// TwinCAT 3 PLC project interlock
// ProgramVersion: 3.1.4023.0
// libraries:
//   VisuElemBase, * (System)
//   Tc2_Standard, * (Beckhoff Automation GmbH)
//   Tc2_System, * (Beckhoff Automation GmbH)
//   Tc3_Module, * (Beckhoff Automation GmbH)
//   Visu Interfaces,newest,System
//   VisuSymbols,3.5.10.0,System
// project tree:
//   / GlobalTextList.TcGTLO, PlcTask.TcTTO, VisualizationManager.TcVMO (not stored), VISU_TASK.TcTTO
//   GVLs/ GVL_ver.TcGVL
//   POUs/ FB_IKR270.TcPOU, FB_KJL300.TcPOU, FB_PBR260.TcPOU, GCC1.TcPOU, GCC2.TcPOU, LadderLogic.TcPOU, LadderLogic_1.TcPOU, MAIN.TcPOU, FB_TCP.TcPOU, VGC1.TcPOU, PTM1.TcPOU, VCC2.TcPOU, VCC3.TcPOU, VGC0.TcPOU
//   VISUs/ Vacuum.TcVIS
// real-time tasks:
//   TASK PlcTask: cycle T#10ms, priority 20, ADS port 350
//   TASK VISU_TASK: cycle T#200000us, priority 30, ADS port 351
// I/O:
//   DEVICE Device 1 (EtherCAT), AmsNetId 5.46.196.210.2.1
//     Term 1 (EK1200) [EK1200-5000 EtherCAT Power supply (2A E-Bus)]
//       Term 2 (EL9210) [EL9210 Power Supplier with LED (24V, Fuse, Diagnostics)]
//       Term 3 (EL3104) [EL3104 4Ch. Ana. Input +/-10V Diff.]
//       Term 4 (EL2004) [EL2004 4Ch. Dig. Output 24V, 0.5A]
//       Term 5 (EL2624) [EL2624 4Ch. Relay Output, NO (125V AC / 30V DC)]
//       Term 6 (EL1104) [EL1104 4Ch. Dig. Input 24V, 3ms, Sensor Power]
//       Term 7 (EL1104) [EL1104 4Ch. Dig. Input 24V, 3ms, Sensor Power]
//       Term 8 (EL2004) [EL2004 4Ch. Dig. Output 24V, 0.5A]
//       Term 9 (EL1104) [EL1104 4Ch. Dig. Input 24V, 3ms, Sensor Power]
//       Term 10 (EL2624) [EL2624 4Ch. Relay Output, NO (125V AC / 30V DC)]
//       Term 11 (EL1104) [EL1104 4Ch. Dig. Input 24V, 3ms, Sensor Power]
//       Term 12 (EL1104) [EL1104 4Ch. Dig. Input 24V, 3ms, Sensor Power]
//       Term 13 (EL2004) [EL2004 4Ch. Dig. Output 24V, 0.5A]
//       Term 14 (EL6022) [EL6022 Interface 2Ch. (RS422/485)]
//       Term 15 (EL6022) [EL6022 Interface 2Ch. (RS422/485)]
//       Term 16 (EK1110) [EK1110 EtherCAT extension]
//   DEVICE Device 3 (CX9020-0115-M310), AmsNetId 5.46.196.210.4.1
//   DEVICE Device 4 (NOV-DP-RAM)
// variable links:
//   interlock Instance <-> Device 1 (EtherCAT)/Term 1 (EK1200)/Term 10 (EL2624)
//     PlcTask Outputs/GVL_ver.VCC2_q_xOPN_DO <-> Channel 1/Output
//   interlock Instance <-> Device 1 (EtherCAT)/Term 1 (EK1200)/Term 12 (EL1104)
//     PlcTask Inputs/GVL_ver.PTM1_i_xAtSpd <-> Channel 1/Input
//     PlcTask Inputs/GVL_ver.PTM1_i_xFaultNC <-> Channel 3/Input
//     PlcTask Inputs/GVL_ver.PTM1_i_xRemote <-> Channel 2/Input
//   interlock Instance <-> Device 1 (EtherCAT)/Term 1 (EK1200)/Term 13 (EL2004)
//     PlcTask Outputs/GVL_ver.PTM1_q_PumpingStation <-> Channel 2/Output
//     PlcTask Outputs/GVL_ver.PTM1_q_RunDO <-> Channel 1/Output
//     PlcTask Outputs/GVL_ver.PTM1_q_xRemote <-> Channel 3/Output
//   interlock Instance <-> Device 1 (EtherCAT)/Term 1 (EK1200)/Term 3 (EL3104)
//     PlcTask Inputs/GVL_ver.GCC1AO <-> AI Standard Channel 1/Value
//     PlcTask Inputs/GVL_ver.GCC2AO <-> AI Standard Channel 2/Value
//   interlock Instance <-> Device 1 (EtherCAT)/Term 1 (EK1200)/Term 4 (EL2004)
//     PlcTask Outputs/GVL_ver.GCC1_xHV_DIS <-> Channel 2/Output
//     PlcTask Outputs/GVL_ver.GCC2_xHV_DIS <-> Channel 4/Output
//   interlock Instance <-> Device 1 (EtherCAT)/Term 1 (EK1200)/Term 6 (EL1104)
//     PlcTask Inputs/GVL_ver.VGC0_i_xClsLS <-> Channel 4/Input
//     PlcTask Inputs/GVL_ver.VGC1_i_xClsLS <-> Channel 3/Input
//     PlcTask Inputs/GVL_ver.VGC0_i_xOpnLS <-> Channel 2/Input
//     PlcTask Inputs/GVL_ver.VGC1_i_xOpnLS <-> Channel 1/Input
//   interlock Instance <-> Device 1 (EtherCAT)/Term 1 (EK1200)/Term 7 (EL1104)
//     PlcTask Inputs/GVL_ver.VCC3_i_xClsLS <-> Channel 4/Input
//     PlcTask Inputs/GVL_ver.VCC3_i_xOpnLS <-> Channel 2/Input
//   interlock Instance <-> Device 1 (EtherCAT)/Term 1 (EK1200)/Term 8 (EL2004)
//     PlcTask Outputs/GVL_ver.VCC3_q_xOPN_DO <-> Channel 4/Output
//     PlcTask Outputs/GVL_ver.VGC0_q_xOPN_DO <-> Channel 3/Output
//     PlcTask Outputs/GVL_ver.VGC1_q_xOPN_DO <-> Channel 1/Output
//   interlock Instance <-> Device 1 (EtherCAT)/Term 1 (EK1200)/Term 9 (EL1104)
//     PlcTask Inputs/GVL_ver.VCC2_i_xClsLS <-> Channel 2/Input
//     PlcTask Inputs/GVL_ver.VCC2_i_xOpnLS <-> Channel 1/Input

CONFIGURATION interlock
    RESOURCE PLC ON TwinCAT3
        TASK PlcTask(INTERVAL := T#10ms, PRIORITY := 20);
        TASK VISU_TASK(INTERVAL := T#200000us, PRIORITY := 30);
        PROGRAM MAIN WITH PlcTask : MAIN;
        PROGRAM VisuElems_Visu_Prg WITH VISU_TASK : VisuElems.Visu_Prg;
    END_RESOURCE
END_CONFIGURATION

// ---- GVLs/GVL_ver.TcGVL
{attribute 'qualified_only'}
VAR_GLOBAL
	V0OPENREQ AT %I*:BOOL;
	V1BYPASS AT %I*:BOOL;
	V2OPENREQ AT %I*:BOOL;
	V3OPENREQ AT %I*:BOOL;
	V4OPENREQ AT %I*:BOOL;
	PTM1STARTREQ AT %I*:BOOL;
	PTM2STARTREQ AT %I*:BOOL;
	PTM3STARTREQ AT %I*:BOOL;
	GCC1ONREQ AT %I*:BOOL;
	GCC2ONREQ AT %I*:BOOL;
	GCC1AO AT %I*:INT;
	GCC2AO AT %I*:INT;

	VGC0OPENREQ AT %I*:BOOL;
	VGC1OPENREQ AT %I*:BOOL;
	VCC2_r_OPENREQ AT %I*:BOOL;
	VCC3_r_OPENREQ AT %I*:BOOL;
	
	PTM1_q_RunDO AT%Q*: BOOL; // Start/Stop for TC110 link this output to the Pumping station bit -3-
    PTM1_q_PumpingStation AT%Q*: BOOL; // Start/Stop interlock -4-
    PTM1_q_xRemote AT%Q*: BOOL; // Remote Priority -14-
    PTM1_i_xAtSpd AT%I*: BOOL; // Normaml operation when true -8-
    PTM1_i_xRemote AT%I*: BOOL; // Remote Priority RBV -23-
	PTM1_i_xFaultNC AT%I*: BOOL; // Error -9-
	
    PTM2_q_RunDO AT%Q*: BOOL; // Start/Stop for TC110 link this output to the Pumping station bit -3-
    PTM2_q_PumpingStation AT%Q*: BOOL; // Start/Stop interlock -4-
    PTM2_q_xRemote AT%Q*: BOOL; // Remote Priority -14-
    PTM2_i_xAtSpd AT%I*: BOOL; // Normaml operation when true -8-
    PTM2_i_xRemote AT%I*: BOOL; // Remote Priority RBV -23-
	PTM2_i_xFaultNC AT%I*: BOOL; // Error -9-
	
	PTM3_q_RunDO AT%Q*: BOOL; // Start/Stop for TC110 link this output to the Pumping station bit -3-
    PTM3_q_PumpingStation AT%Q*: BOOL; // Start/Stop interlock -4-
    PTM3_q_xRemote AT%Q*: BOOL; // Remote Priority -14-
    PTM3_i_xAtSpd AT%I*: BOOL; // Normaml operation when true -8-
    PTM3_i_xRemote AT%I*: BOOL; // Remote Priority RBV -23-
	PTM3_i_xFaultNC AT%I*: BOOL; // Error -9-
	
	VGC0_q_xOPN_DO AT%Q*: BOOL; //24V open/close
	VGC0_i_xOpnLS AT%I*  : BOOL; //Open position SW
    VGC0_i_xClsLS AT%I*  : BOOL; //Close position SW
	VGC0_i_xUpstream_OK  AT%Q*  : BOOL;
	VGC0_i_xDwstream_OK  AT%Q*  : BOOL;
	
	VGC1_q_xOPN_DO AT%Q*: BOOL; //24V open/close
	VGC1_i_xOpnLS AT%I*  : BOOL; //Open position SW
    VGC1_i_xClsLS AT%I*  : BOOL; //Close position SW
	VGC1_i_xUpstream_OK  AT%Q*  : BOOL;
	VGC1_i_xDwstream_OK  AT%Q*  : BOOL;
    
    VCC2_q_xOPN_DO AT%Q*: BOOL; //24V open/close
	VCC2_i_xOpnLS AT%I*  : BOOL; //Open position SW
    VCC2_i_xClsLS AT%I*  : BOOL; //Close position SW
    
    VCC3_q_xOPN_DO AT%Q*: BOOL; //24V open/close
	VCC3_i_xOpnLS AT%I*  : BOOL; //Open position SW
    VCC3_i_xClsLS AT%I*  : BOOL; //Close position SW
    
    GCC1_rPRESS AT%Q* : REAL; //This is the human-readable pressure
    GCC1_xPRESS_OK AT%Q*: BOOL;
	GCC1_xHV_DIS AT %Q* : BOOL;
	
	GCC2_rPRESS AT%Q*: REAL; //This is the human-readable pressure
    GCC2_xPRESS_OK AT%Q*: BOOL;
	GCC2_xHV_DIS AT %Q* : BOOL;

END_VAR

// ---- POUs/MAIN.TcPOU
PROGRAM MAIN
VAR
END_VAR

GVL_ver.GCC2_xHV_DIS:=TRUE;
LadderLogic();
FB_KJL300();
FB_PBR260();
FB_TCP();

END_PROGRAM

// ---- POUs/LadderLogic.TcPOU
PROGRAM LadderLogic
VAR
	ExternalILK: BOOL;
END_VAR

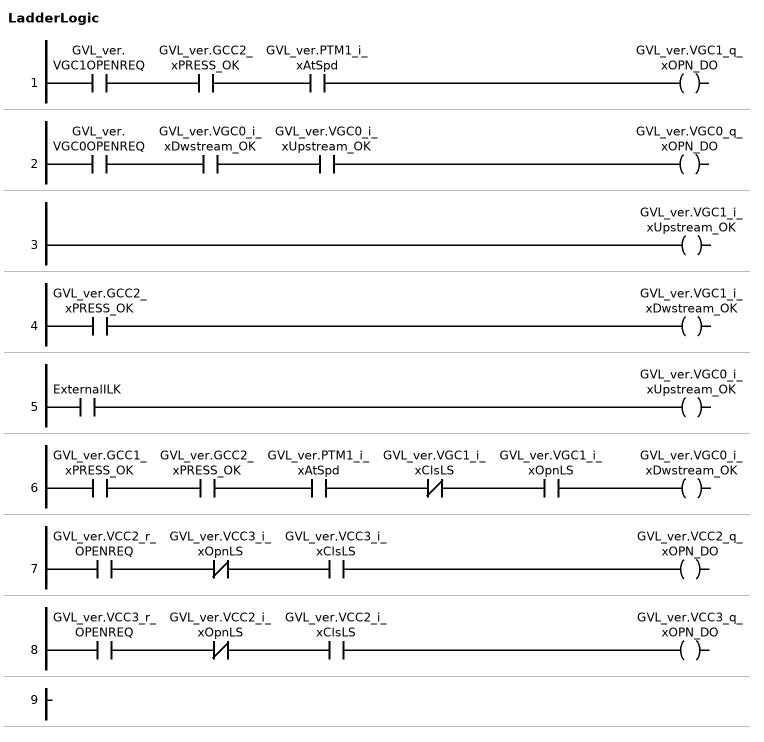
// NETWORK 1
GVL_ver.VGC1_q_xOPN_DO := GVL_ver.VGC1OPENREQ AND GVL_ver.GCC2_xPRESS_OK AND GVL_ver.PTM1_i_xAtSpd;

// NETWORK 2
GVL_ver.VGC0_q_xOPN_DO := GVL_ver.VGC0OPENREQ AND GVL_ver.VGC0_i_xDwstream_OK AND GVL_ver.VGC0_i_xUpstream_OK;

// NETWORK 3
GVL_ver.VGC1_i_xUpstream_OK := TRUE;

// NETWORK 4
GVL_ver.VGC1_i_xDwstream_OK := GVL_ver.GCC2_xPRESS_OK;

// NETWORK 5
GVL_ver.VGC0_i_xUpstream_OK := ExternalILK;

// NETWORK 6
GVL_ver.VGC0_i_xDwstream_OK := GVL_ver.GCC1_xPRESS_OK AND GVL_ver.GCC2_xPRESS_OK AND GVL_ver.PTM1_i_xAtSpd AND NOT GVL_ver.VGC1_i_xClsLS AND GVL_ver.VGC1_i_xOpnLS;

// NETWORK 7
GVL_ver.VCC2_q_xOPN_DO := GVL_ver.VCC2_r_OPENREQ AND NOT GVL_ver.VCC3_i_xOpnLS AND GVL_ver.VCC3_i_xClsLS;

// NETWORK 8
GVL_ver.VCC3_q_xOPN_DO := GVL_ver.VCC3_r_OPENREQ AND NOT GVL_ver.VCC2_i_xOpnLS AND GVL_ver.VCC2_i_xClsLS;

// NETWORK 9

END_PROGRAM

// ---- POUs/FB_KJL300.TcPOU
PROGRAM FB_KJL300
VAR
	AO:INT;
	rPRESS:REAL;
	xPRESS_OK:BOOL;
	xHV_DIS:BOOL:=TRUE;
END_VAR

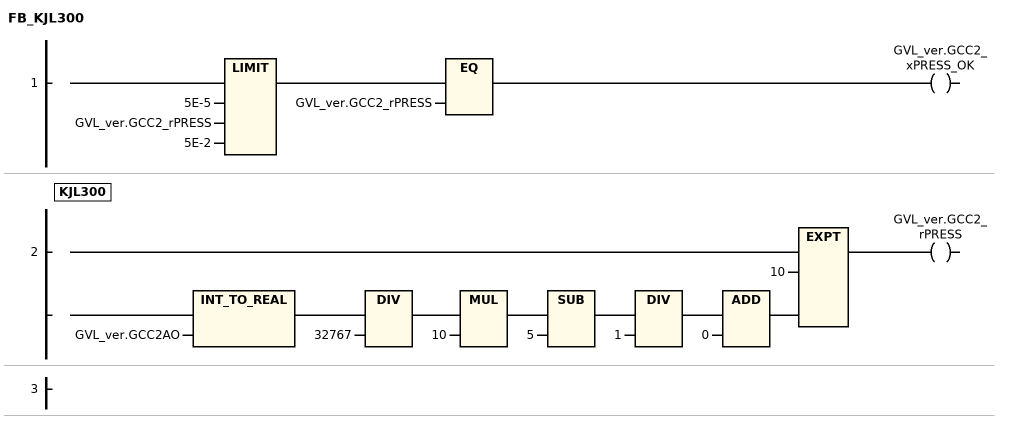
// NETWORK 1
GVL_ver.GCC2_xPRESS_OK := LIMIT(5E-5, GVL_ver.GCC2_rPRESS, 5E-2) = GVL_ver.GCC2_rPRESS;

// NETWORK 2
KJL300:
GVL_ver.GCC2_rPRESS := EXPT(10, ((INT_TO_REAL(GVL_ver.GCC2AO) / 32767) * 10 - 5) / 1 + 0);

// NETWORK 3

END_PROGRAM

// ---- POUs/FB_PBR260.TcPOU
PROGRAM FB_PBR260
VAR
	AO:INT;
	rPRESS:REAL;
	xPRESS_OK:BOOL;
	xHV_DIS:BOOL;
END_VAR

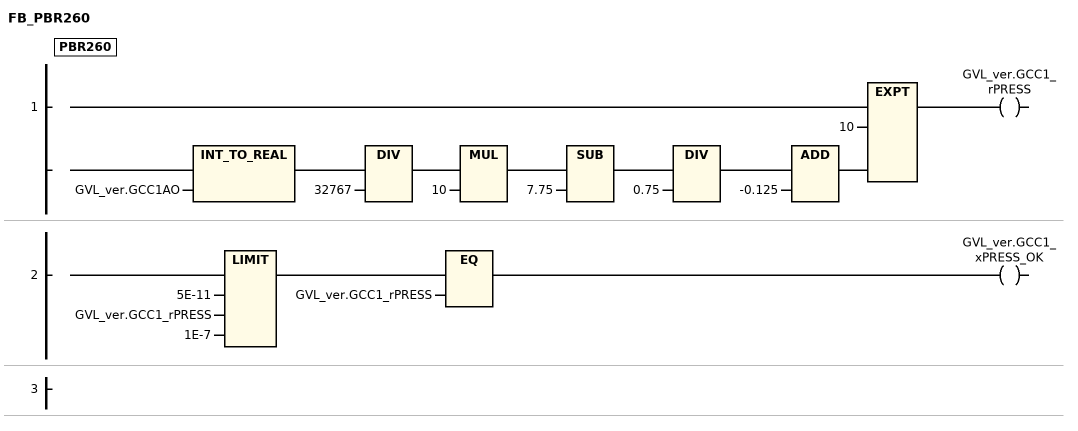
// NETWORK 1
PBR260:
GVL_ver.GCC1_rPRESS := EXPT(10, ((INT_TO_REAL(GVL_ver.GCC1AO) / 32767) * 10 - 7.75) / 0.75 + -0.125);

// NETWORK 2
GVL_ver.GCC1_xPRESS_OK := LIMIT(5E-11, GVL_ver.GCC1_rPRESS, 1E-7) = GVL_ver.GCC1_rPRESS;

// NETWORK 3

END_PROGRAM

// ---- POUs/FB_TCP.TcPOU
PROGRAM FB_TCP
VAR
END_VAR
VAR // added by the converter: edge detectors and wires of the graphical bodies
    _w1 : BOOL;
END_VAR

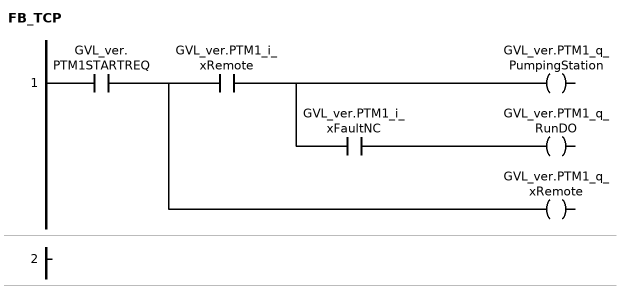
// NETWORK 1
_w1 := GVL_ver.PTM1STARTREQ AND GVL_ver.PTM1_i_xRemote;
GVL_ver.PTM1_q_PumpingStation := _w1;
GVL_ver.PTM1_q_RunDO := _w1 AND GVL_ver.PTM1_i_xFaultNC;
GVL_ver.PTM1_q_xRemote := GVL_ver.PTM1STARTREQ;

// NETWORK 2

END_PROGRAM

// ---- POUs/FB_IKR270.TcPOU
PROGRAM FB_IKR270
VAR
	AO:INT;
	rPRESS:REAL;
	xPRESS_OK:BOOL;
	xHV_DIS:BOOL;
END_VAR

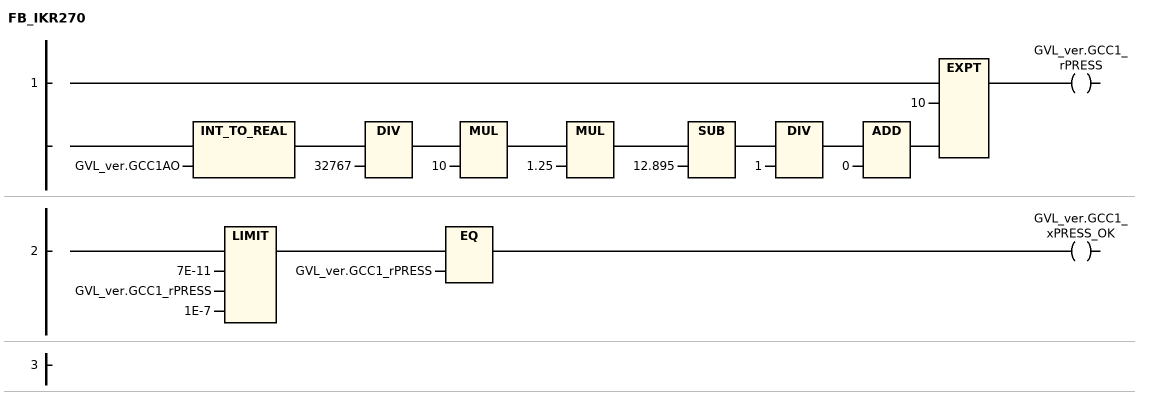
// NETWORK 1
GVL_ver.GCC1_rPRESS := EXPT(10, (((INT_TO_REAL(GVL_ver.GCC1AO) / 32767) * 10) * 1.25 - 12.895) / 1 + 0);

// NETWORK 2
GVL_ver.GCC1_xPRESS_OK := LIMIT(7E-11, GVL_ver.GCC1_rPRESS, 1E-7) = GVL_ver.GCC1_rPRESS;

// NETWORK 3

END_PROGRAM

// ---- POUs/GCC1.TcPOU
PROGRAM GCC1
VAR
END_VAR

// NETWORK 1

END_PROGRAM

// ---- POUs/GCC2.TcPOU
PROGRAM GCC2
VAR
END_VAR

END_PROGRAM

// ---- POUs/LadderLogic_1.TcPOU
PROGRAM LadderLogic_1
VAR
END_VAR
VAR // added by the converter: edge detectors and wires of the graphical bodies
    _w1, _w2, _w3 : BOOL;
END_VAR

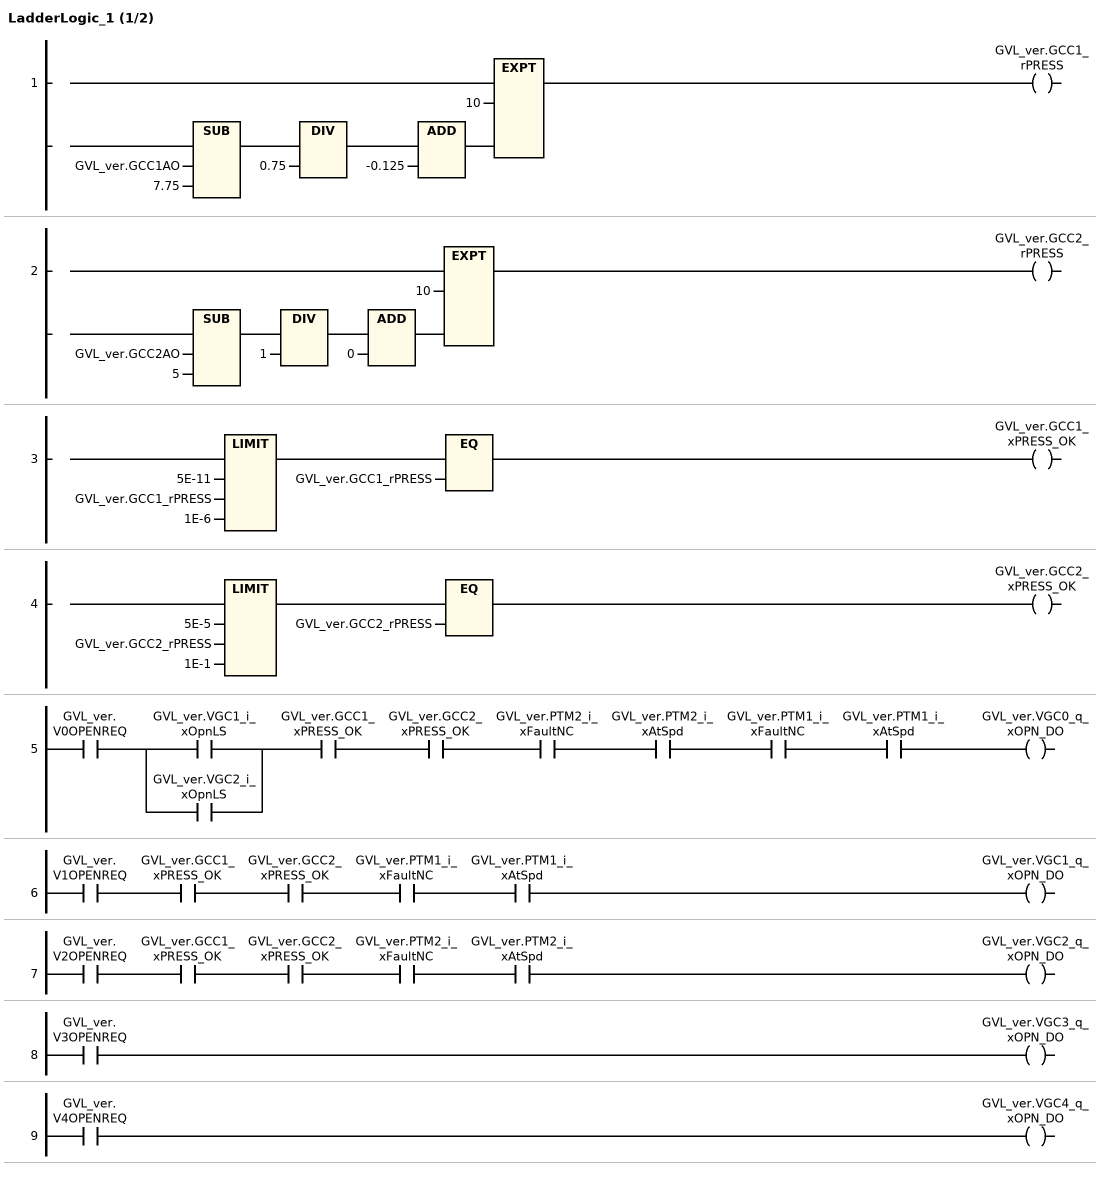
// NETWORK 1
GVL_ver.GCC1_rPRESS := EXPT(10, (GVL_ver.GCC1AO - 7.75) / 0.75 + -0.125);

// NETWORK 2
GVL_ver.GCC2_rPRESS := EXPT(10, (GVL_ver.GCC2AO - 5) / 1 + 0);

// NETWORK 3
GVL_ver.GCC1_xPRESS_OK := LIMIT(5E-11, GVL_ver.GCC1_rPRESS, 1E-6) = GVL_ver.GCC1_rPRESS;

// NETWORK 4
GVL_ver.GCC2_xPRESS_OK := LIMIT(5E-5, GVL_ver.GCC2_rPRESS, 1E-1) = GVL_ver.GCC2_rPRESS;

// NETWORK 5
GVL_ver.VGC0_q_xOPN_DO := GVL_ver.V0OPENREQ AND (GVL_ver.VGC1_i_xOpnLS OR GVL_ver.VGC2_i_xOpnLS) AND GVL_ver.GCC1_xPRESS_OK AND GVL_ver.GCC2_xPRESS_OK AND GVL_ver.PTM2_i_xFaultNC AND GVL_ver.PTM2_i_xAtSpd AND GVL_ver.PTM1_i_xFaultNC AND GVL_ver.PTM1_i_xAtSpd;

// NETWORK 6
GVL_ver.VGC1_q_xOPN_DO := GVL_ver.V1OPENREQ AND GVL_ver.GCC1_xPRESS_OK AND GVL_ver.GCC2_xPRESS_OK AND GVL_ver.PTM1_i_xFaultNC AND GVL_ver.PTM1_i_xAtSpd;

// NETWORK 7
GVL_ver.VGC2_q_xOPN_DO := GVL_ver.V2OPENREQ AND GVL_ver.GCC1_xPRESS_OK AND GVL_ver.GCC2_xPRESS_OK AND GVL_ver.PTM2_i_xFaultNC AND GVL_ver.PTM2_i_xAtSpd;

// NETWORK 8
GVL_ver.VGC3_q_xOPN_DO := GVL_ver.V3OPENREQ;

// NETWORK 9
GVL_ver.VGC4_q_xOPN_DO := GVL_ver.V4OPENREQ;

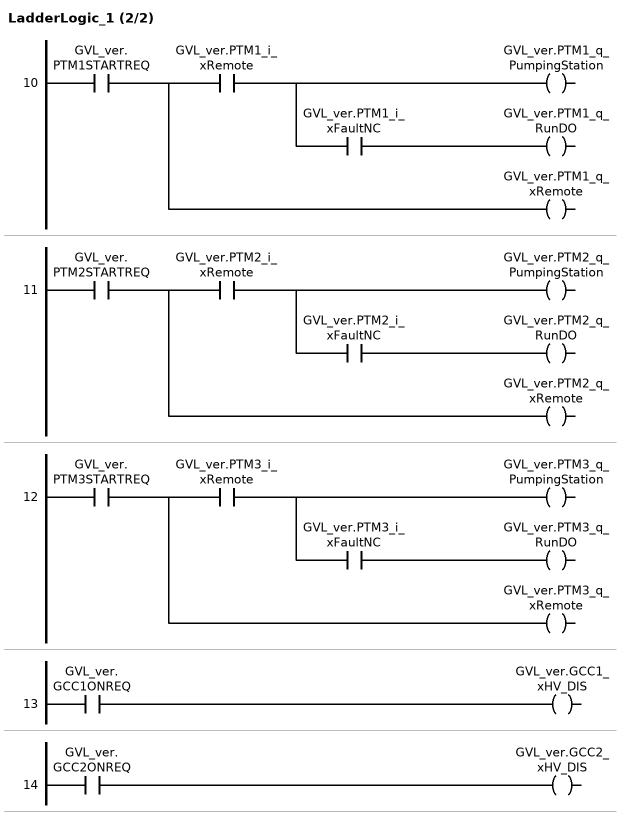
// NETWORK 10
_w1 := GVL_ver.PTM1STARTREQ AND GVL_ver.PTM1_i_xRemote;
GVL_ver.PTM1_q_PumpingStation := _w1;
GVL_ver.PTM1_q_RunDO := _w1 AND GVL_ver.PTM1_i_xFaultNC;
GVL_ver.PTM1_q_xRemote := GVL_ver.PTM1STARTREQ;

// NETWORK 11
_w2 := GVL_ver.PTM2STARTREQ AND GVL_ver.PTM2_i_xRemote;
GVL_ver.PTM2_q_PumpingStation := _w2;
GVL_ver.PTM2_q_RunDO := _w2 AND GVL_ver.PTM2_i_xFaultNC;
GVL_ver.PTM2_q_xRemote := GVL_ver.PTM2STARTREQ;

// NETWORK 12
_w3 := GVL_ver.PTM3STARTREQ AND GVL_ver.PTM3_i_xRemote;
GVL_ver.PTM3_q_PumpingStation := _w3;
GVL_ver.PTM3_q_RunDO := _w3 AND GVL_ver.PTM3_i_xFaultNC;
GVL_ver.PTM3_q_xRemote := GVL_ver.PTM3STARTREQ;

// NETWORK 13
GVL_ver.GCC1_xHV_DIS := GVL_ver.GCC1ONREQ;

// NETWORK 14
GVL_ver.GCC2_xHV_DIS := GVL_ver.GCC2ONREQ;

END_PROGRAM

// ---- POUs/VGC1.TcPOU
PROGRAM VGC1
VAR
END_VAR

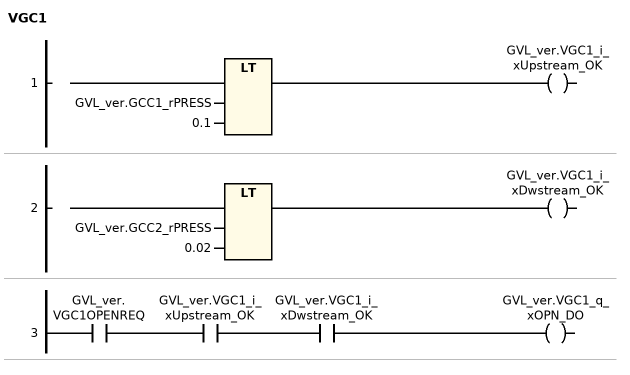
// NETWORK 1
GVL_ver.VGC1_i_xUpstream_OK := GVL_ver.GCC1_rPRESS < 0.1;

// NETWORK 2
GVL_ver.VGC1_i_xDwstream_OK := GVL_ver.GCC2_rPRESS < 0.02;

// NETWORK 3
GVL_ver.VGC1_q_xOPN_DO := GVL_ver.VGC1OPENREQ AND GVL_ver.VGC1_i_xUpstream_OK AND GVL_ver.VGC1_i_xDwstream_OK;

END_PROGRAM

// ---- POUs/PTM1.TcPOU
PROGRAM PTM1
VAR
END_VAR

END_PROGRAM

// ---- POUs/VCC2.TcPOU
PROGRAM VCC2
VAR
END_VAR

END_PROGRAM

// ---- POUs/VCC3.TcPOU
PROGRAM VCC3
VAR
END_VAR

END_PROGRAM

// ---- POUs/VGC0.TcPOU
PROGRAM VGC0
VAR
END_VAR

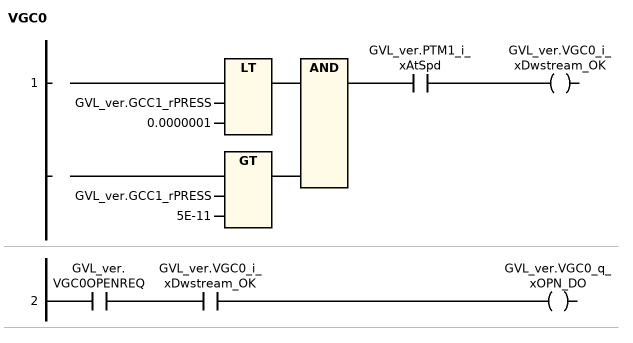
// NETWORK 1
GVL_ver.VGC0_i_xDwstream_OK := (GVL_ver.GCC1_rPRESS < 0.0000001 AND GVL_ver.GCC1_rPRESS > (5E-11)) AND GVL_ver.PTM1_i_xAtSpd;

// NETWORK 2
GVL_ver.VGC0_q_xOPN_DO := GVL_ver.VGC0OPENREQ AND GVL_ver.VGC0_i_xDwstream_OK;

END_PROGRAM

// ---- GlobalTextList.TcGTLO
TEXTLIST GlobalTextList
  953 = '%.3e'
  559 = '%d'
  594 = '%d*'
  835 = 'AtSpd'
  251 = 'Beamline'
  163 = 'BL'
  153 = 'CL Main Turbo Valve OP'
  40 = 'CLOSED'
  723 = 'End Station'
  312 = 'FaultNC'
  47 = 'GCC1'
  977 = 'GCC1 & TPM1 & GCC2'
  613 = 'GCC2'
  874 = 'Main TPM1 '
  833 = 'Main Turbo 400'
  959 = 'Main Turbo 80'
  225 = 'Main Turbo TPM1'
  734 = 'Main Turbo TPM1 RMT'
  854 = 'Main Turbo TPM1 Rremote'
  443 = 'Main Turbo Valve'
  763 = 'OP BL Valve CL'
  728 = 'OP BL VGC CL'
  124 = 'OP BL VGC0 CL'
  642 = 'OP Main Turbo Valve CL'
  794 = 'OP Main Turbo VCC CL'
  638 = 'OP Main Turbo VCC2 CL'
  199 = 'OP Main Turbo VCL'
  480 = 'OP Main Turbo VGC CL'
  41 = 'OP Main Turbo VGC1 CL'
  687 = 'OP Main Turbo VGG CL'
  845 = 'OP Main Turbo VPG CL'
  599 = 'OP Small Turbo VCC CL'
  992 = 'OP Small Turbo VCC3 CL'
  806 = 'OP Turbo Valve CL'
  111 = 'OPEN'
  333 = 'OPN_DO'
  621 = 'PRESS_OK'
  414 = 'RESS_OK'
  226 = 'Small TPM2'
  801 = 'Small TPM2 RMT'
  297 = 'Small TPM3'
  383 = 'Small TPM3 Remote'
  676 = 'Small TPM3 RMT'
  840 = 'Small Trubo 80'
  159 = 'Small Trubo TPM2'
  611 = 'Small Trubo TPM2 RMT'
  175 = 'T'
  899 = 'TPM01 Start/Stop'
  715 = 'TPM1'
  629 = 'TPM2'
  51 = 'TPM3'
  172 = 'VGC0'
  550 = 'VGC01'
  274 = 'VGC1'
  384 = 'VGC2'
  171 = 'VGC3'
  221 = 'VGC4'
END_TEXTLIST

// ---- VISUs/Vacuum.TcVIS
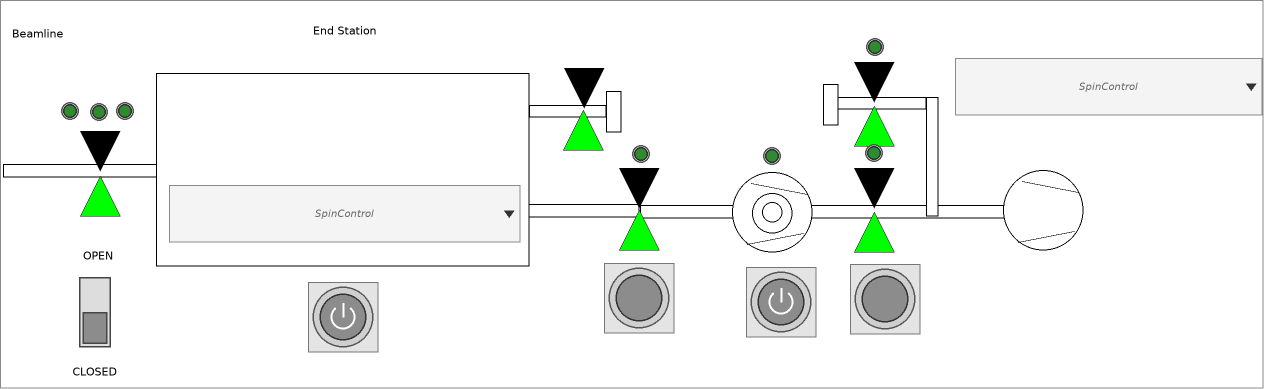
VISUALIZATION Vacuum  // 1264x389
    Rectangle (529,105 77x12)
    Rectangle (640,205 380x13), colour toggle: GVL_ver.VGC1_i_xDwstream_OK
    Rectangle (523,204 116x13), colour toggle: GVL_ver.VGC1_i_xUpstream_OK
    Rectangle (3,164 467x13)
    RoundedRectangle (156,73 373x193), colour toggle: GVL_ver.GCC1_xPRESS_OK
    SpinControl (169,185 351x57), variable: GVL_ver.GCC1_rPRESS
    SpinControl (955,58 307x57), variable: GVL_ver.GCC2_rPRESS
    PowerSwitch (308,282 70x70), variable: GVL_ver.GCC1_xHV_DIS, behaviour: TOGGLE, style: Switch-PowerSwitch-Gray
    PushSwitchLed (604,263 70x70), variable: GVL_ver.VGC1OPENREQ, behaviour: TOGGLE, style: Switch-PushSwitchLed-Gray
    Lamp1 (762,146 20x20), variable: GVL_ver.PTM1_i_xFaultNC, style: Lamp-Lamp1-Green
    PowerSwitch (746,267 70x70), variable: GVL_ver.PTM1STARTREQ, behaviour: TOGGLE, style: Switch-PowerSwitch-Gray
    Polygon (639,210) (639,210) (639,210) (659,250) (619,250), colour toggle: GVL_ver.VGC1_i_xClsLS
    Polygon (639,208) (639,208) (639,208) (659,168) (619,168), colour toggle: GVL_ver.VGC1_i_xOpnLS
    Ellipse (732,172 80x80), colour toggle: GVL_ver.PTM1_i_xAtSpd
    Ellipse (752,193 40x40), colour toggle: GVL_ver.PTM1_q_RunDO
    Ellipse (762,202 20x20), colour toggle: GVL_ver.PTM1_q_PumpingStation
    Polygon (874,208) (874,208) (874,208) (894,168) (854,168), colour toggle: GVL_ver.VCC2_i_xOpnLS
    Polygon (583,110) (583,110) (583,110) (603,150) (563,150), colour toggle: GVL_ver.VCC3_i_xClsLS
    PushSwitchLed (850,264 70x70), variable: GVL_ver.VCC2_r_OPENREQ, behaviour: TOGGLE, style: Switch-PushSwitchLed-Gray
    Line (822,135)
    Line (747,244) (803,233), colour toggle: GVL_ver.PTM1_q_xRemote
    Line (751,183) (807,194), colour toggle: GVL_ver.PTM1_i_xRemote
    Polygon (584,108) (584,108) (584,108) (604,68) (564,68), colour toggle: GVL_ver.VCC3_i_xOpnLS
    Rectangle (606,91 15x41)
    Polygon (100,171) (100,171) (100,171) (120,131) (80,131), colour toggle: GVL_ver.VGC0_i_xOpnLS
    Polygon (100,176) (100,176) (100,176) (120,216) (80,216), colour toggle: GVL_ver.VGC0_i_xClsLS
    Polygon (874,212) (874,212) (874,212) (894,252) (854,252), colour toggle: GVL_ver.VCC2_i_xClsLS
    Rectangle (824,97 102x12), colour toggle: GVL_ver.VGC1_i_xDwstream_OK
    Polygon (874,106) (874,106) (874,106) (894,146) (854,146), colour toggle: GVL_ver.VCC3_i_xClsLS
    Polygon (874,102) (874,102) (874,102) (894,62) (854,62), colour toggle: GVL_ver.VCC3_i_xOpnLS
    DipSwitch (60,277 70x70), variable: GVL_ver.VGC0OPENREQ, behaviour: TOGGLE, style: Switch-DipSwitch-Gray
    Label (63,241 70x30), "OPEN"
    Label (60,357 70x30), "CLOSED"
    Ellipse (1003,170 80x80), colour toggle: GVL_ver.PTM2_i_xAtSpd
    Line (1018,242) (1074,231), colour toggle: GVL_ver.PTM1_q_xRemote
    Line (1022,181) (1078,192), colour toggle: GVL_ver.PTM1_i_xRemote
    Rectangle (926,97 12x119), colour toggle: GVL_ver.VGC1_i_xDwstream_OK
    Rectangle (823,84 15x41)
    Label (3,19 70x30), "Beamline"
    Label (295,16 100x30), "End Station"
    Lamp1 (631,144 20x20), variable: GVL_ver.VGC1_q_xOPN_DO, style: Lamp-Lamp1-Green
    Lamp1 (89,102 20x20), variable: GVL_ver.VGC0_q_xOPN_DO, style: Lamp-Lamp1-Green
    Lamp1 (115,101 20x20), variable: GVL_ver.VGC0_i_xDwstream_OK, style: Lamp-Lamp1-Green
    Lamp1 (60,101 20x20), variable: GVL_ver.VGC0_i_xUpstream_OK, style: Lamp-Lamp1-Green
    Lamp1 (864,143 20x20), variable: GVL_ver.VCC2_q_xOPN_DO, style: Lamp-Lamp1-Green
    Lamp1 (865,37 20x20), variable: GVL_ver.VCC3_q_xOPN_DO, style: Lamp-Lamp1-Green
END_VISUALIZATION
